//Test GVL
{attribute 'qualified_only'}
VAR_GLOBAL
END_VAR

(* stored: Version 1.1.0.1, ProductVersion 3.1.4024.12
   GVL GVL_Sys: Id {4e67ab74-6b7c-4b72-803a-1e3548a94041} *)
